	    REGION Part_MC_to_Robot
	        CASE #Dispatcher["_Part_MC_to_Robot"] OF
	            0: //nothing to do
	                ;
	            10: //prepare mission data
	                IF "SqlCommands".sqlCommands[0] = '' THEN
	                    IF #Gripper_ID[1] = 0 AND #Gripper_ID[2] = 0 THEN
	                        //nessuna pinza a bordo: impossibile prelevare
	                        #Error := 16;
	                        #Dispatcher["_Part_MC_to_Robot"] := "_Part_MC_to_Robot" * 100 + 1;
	                    ELSIF #GripperOccuped[1] AND #GripperOccuped[2] THEN
	                        //nessun lato libero: impossibile prelevare
	                        #Error := 18;
	                        #Dispatcher["_Part_MC_to_Robot"] := "_Part_MC_to_Robot" * 100 + 1;
	                    ELSIF (#MCRequested = 1 AND "DB_MC1".io_in.viceOpened) THEN
	                        // MORSA APERTA = NESSUN PEZZO DA PRELEVARE (17/9).
	                        // La ganascia aperta non puo' trattenere niente: qualunque
	                        // cosa dicano i registri, in morsa non c'e' un pezzo. Il
	                        // contrario NON vale — chiusa non implica pieno, puo'
	                        // essersi chiusa a vuoto — quindi il segnale si usa solo
	                        // come VETO, mai come conferma.
	                        #Error := 894;
	                        #Dispatcher["_Part_MC_to_Robot"] := 894;
	                    ELSE
	                        // QUOTE DALLA VISTA COORDINATES_Z_MC (19/9): vedi nota al
	                        // 10 di Part_Robot_to_MC.
	                        // Z_PICK_MC = prelievo del FINITO, che puo' avere presa
	                        // diversa dal grezzo (15/9).
	                        #queryTemp := 'select P.X,P.Y,Z.Z_PICK_MC,P.X_ROT,P.Y_ROT,P.Z_ROT,P.APPROACH_TYPE,P.APPROACH_X,P.APPROACH_Y,P.APPROACH_Z from POSITION P,COORDINATES_Z_MC Z where P.PARENT=$'MC_1$' and ';
	                        IF #RemoteMode THEN
	                            IF #MCRequested = 1 AND "DB_MC1".order.ID > 0 THEN
	                                #queryTemp := CONCAT(IN1 := #queryTemp,
	                                                     IN2 := 'Z.ORDER_ID=',
	                                                     IN3 := "INT_TO_STRING_WITHOUT_SIGN"(DINT_TO_INT("DB_MC1".order.ID)));
	                            ELSE
	                                #Error := 936;
	                                #Dispatcher["_Part_MC_to_Robot"] := "_Part_MC_to_Robot" * 100 + 1;
	                            END_IF;
	                        ELSE
	                            // HMI (29): ordine attivo se presente, altrimenti il piu' recente
	                            IF "DB_MC1".order.ID > 0 THEN
	                                #queryTemp := CONCAT(IN1 := #queryTemp,
	                                                     IN2 := 'Z.ORDER_ID=',
	                                                     IN3 := "INT_TO_STRING_WITHOUT_SIGN"(DINT_TO_INT("DB_MC1".order.ID)));
	                            ELSE
	                                #queryTemp := CONCAT(IN1 := #queryTemp,
	                                                     IN2 := 'Z.MC=1 order by Z.ORDER_ID desc');
	                            END_IF;
	                        END_IF;

	                        IF #Error = 0 THEN
	                            #queryStartExecution := TRUE;
	                            #Dispatcher["_Part_MC_to_Robot"] := 20;
	                        END_IF;
	                    END_IF;
	                END_IF;

	            20:  //execute query
	                // PRESA IN CARICO VERIFICATA: SqlData e' un buffer unico condiviso,
	                // senza il confronto su sqlCommands[0] si legge la risposta di un
	                // altro richiedente — qui sarebbero le QUOTE DI PRELIEVO dalla morsa.
	                IF NOT "DB_executeQuery".readyForNextQuery
	                    AND "SqlCommands".sqlCommands[0] = #queryTemp THEN
	                    #Dispatcher["_Part_MC_to_Robot"] := 30;
	                END_IF;

	            30:  // wait for result DB -> prepare mission data
	                IF "DB_executeQuery".dataReady AND "DB_executeQuery".noData THEN
	                    // quote di prelievo non trovate: con FB6 corretto "zero righe"
	                    // non e' piu' dataError, va intercettato qui.
	                    "DB_executeQuery".readyForNextQuery := true;
	                    #Error := "_Part_MC_to_Robot" * 100 + 99;       //Error 899
	                    #Dispatcher["_Part_MC_to_Robot"] := "_Part_MC_to_Robot" * 100 + 99;
	                ELSIF "DB_executeQuery".dataReady AND NOT "DB_executeQuery".dataError THEN

	                    // X DI PRELIEVO + CORSA DELLA SPINTA: se il pezzo e' stato
	                    // spinto in battuta non sta piu' dove il deposito lo ha messo.
	                    // xPushOffsetMC vale zero quando la spinta non c'e' stata,
	                    // quindi il caso normale resta invariato.
	                    "DB_RobotMission"."X_Pick-Place" := ("SqlData".data.rows[0].col[0]) + #xPushOffsetMC;
	                    "DB_RobotMission"."Y_Pick-Place" := ("SqlData".data.rows[0].col[1]);
	                    "DB_RobotMission"."Z_Pick-Place" := ("SqlData".data.rows[0].col[2]);
	                    "DB_RobotMission"."XRot_Pick-Place" := ("SqlData".data.rows[0].col[3]);
	                    "DB_RobotMission"."YRot_Pick-Place" := ("SqlData".data.rows[0].col[4]);
	                    "DB_RobotMission"."ZRot_Pick-Place" := ("SqlData".data.rows[0].col[5]);
	                    "DB_RobotMission".X_approach := ("SqlData".data.rows[0].col[7]);
	                    "DB_RobotMission".Y_approach := ("SqlData".data.rows[0].col[8]);
	                    "DB_RobotMission".Z_approach := ("SqlData".data.rows[0].col[9]);
	                    "DB_RobotMission".XRot_approach := 0;
	                    "DB_RobotMission".YRot_approach := 0;
	                    "DB_RobotMission".ZRot_approach := 0;
	                    //"DB_RobotMission".ApproachType := DINT_TO_INT("SqlData".data.rows[0].col[6]);
	                    "DB_RobotMission".ApproachType := "FC_ExtractApproach"(approachVal := "SqlData".data.rows[0].col[6], pick := TRUE);
	                    "DB_RobotMission".Object_Type := "Part";
	                    "DB_RobotMission".Unit_code := #MCRequested + 10;
	                    "DB_RobotMission".Gripper_code := #GripperRequested;
	                    // LATO SEMPRE DECISO (5/10): mancava l'ELSE. Con la doppia e il lato 2
	                    // pieno, o con la singola piena, Gripper_Side restava quello della
	                    // missione precedente e il robot prelevava con un lato occupato. Il lato
	                    // 1 della doppia e' del grezzo: il finito non ci va.
	                    "DB_executeQuery".readyForNextQuery := true;
	                    IF (#Gripper_ID[2] <> 0 AND NOT #GripperOccuped[2]) THEN
	                        "DB_RobotMission".Gripper_Side := 2;
	                        #Dispatcher["_Part_MC_to_Robot"] := 37;
	                    ELSIF (#Gripper_ID[2] = 0 AND #Gripper_ID[1] <> 0 AND NOT #GripperOccuped[1]) THEN
	                        "DB_RobotMission".Gripper_Side := 1;
	                        #Dispatcher["_Part_MC_to_Robot"] := 37;
	                    ELSE
	                        #Error := 18;   // nessun lato libero adatto al finito
	                        #Dispatcher["_Part_MC_to_Robot"] := "_Part_MC_to_Robot" * 100 + 1;
	                    END_IF;
	                    //"DB_RobotMission".Option
	                ELSIF "DB_executeQuery".dataError THEN
	                    "DB_executeQuery".readyForNextQuery := true;

	                    //Errore
	                    #Error := "_Part_MC_to_Robot" * 100 + 99;       //Error 899
	                    #Dispatcher["_Part_MC_to_Robot"] := "_Part_MC_to_Robot" * 100 + 99;
	                END_IF;

	            37:  // SOFFIAGGIO: vedi nota estesa al 37 di Part_Robot_to_MC.
	                // NB: qui X_Pick-Place e' la quota di PRELIEVO, che include
	                // xPushOffsetMC se il pezzo e' stato spinto. L'appoggio va
	                // calcolato sulla quota di DEPOSITO, quindi si sottrae l'offset
	                // per tornare alla nominale.
	                IF "SqlCommands".sqlCommands[0] = '' THEN
	                    IF "DB_MC1".order.ID > 0 THEN
	                        #queryTemp := CONCAT(IN1 := 'select CLAW_LENGTH,PART_WIDTH,STOP_BEYOND_CLAW from COORDINATES_BLOW_MC where ORDER_ID=',
	                                             IN2 := "INT_TO_STRING_WITHOUT_SIGN"(DINT_TO_INT("DB_MC1".order.ID)));
	                        #queryStartExecution := TRUE;
	                        #Dispatcher["_Part_MC_to_Robot"] := 38;
	                    ELSE
	                        #Dispatcher["_Part_MC_to_Robot"] := 40;
	                    END_IF;
	                END_IF;

	            38:  // presa in carico VERIFICATA
	                IF NOT "DB_executeQuery".readyForNextQuery
	                    AND "SqlCommands".sqlCommands[0] = #queryTemp THEN
	                    #Dispatcher["_Part_MC_to_Robot"] := 39;
	                END_IF;

	            39:  // esito: scrive le tre variabili PROFINET.
	                // APPOGGIO COME MISURA, NON COME QUOTA (19/9): il robotista non
	                // vuole piu' la posizione X del pezzo, che calcola per conto suo —
	                // gli serve solo di quanto il pezzo appoggia, cioe' meta' ganascia
	                // piu' il tratto oltre la ganascia dichiarato a pannello.
	                // Niente X_Pick-Place e niente xPushOffsetMC: l'offset serviva a
	                // riportare la quota di prelievo a quella di deposito, e senza la
	                // quota non ha piu' nulla da correggere. Sottraendolo dopo la
	                // divisione, per giunta, si toglievano MICRON da un numero in
	                // MILLIMETRI: col push attivo dava -49650.
	                IF "DB_executeQuery".dataReady THEN
	                    IF NOT "DB_executeQuery".noData AND NOT "DB_executeQuery".dataError THEN
	                        "Vice_ClawLength_mm" := DINT_TO_INT("SqlData".data.rows[0].col[0] / 1000);
	                        "Part_Width_mm" := DINT_TO_INT("SqlData".data.rows[0].col[1] / 1000);
	                        "X_Support_mm" := DINT_TO_INT(("SqlData".data.rows[0].col[0] / 2
	                                                                                    + "SqlData".data.rows[0].col[2]) / 1000);
	                    END_IF;
	                    "DB_executeQuery".readyForNextQuery := TRUE;
	                    #queryTemp := '';
	                    #queryStartExecution := FALSE;
	                    #Dispatcher["_Part_MC_to_Robot"] := 40;
	                END_IF;

	            40:
	                "DB_RobotMission".Command := "CMD_RobotPickObject";
	                IF "DB_RobotMissionStatus".StatusCode = "cmd_acquired" OR
	                    "DB_RobotMissionStatus".StatusCode = "cmd_executing" THEN
	                    #Dispatcher["_Part_MC_to_Robot"] := 50;
	                END_IF;
	            50:
	                IF "DB_RobotMissionStatus".StatusCode = "cmd_executed" THEN
	                    // lati dedicati: marca il lato realmente scelto (Gripper_Side: 1=grezzo, 2=finito)
	                    IF "DB_RobotMission".Gripper_Side = 2 THEN
	                        #GripperOccuped[2] := TRUE;
	                        #Dispatcher["updatePartOnRobot"] := 20 + DINT_TO_INT("FINISHED");
	                    ELSE
	                        #GripperOccuped[1] := TRUE;
	                        #Dispatcher["updatePartOnRobot"] := 10 + DINT_TO_INT("FINISHED");
	                    END_IF;
	                    "DB_RobotMission".Command := 0; ///\\\

	                    // Il pezzo spinto e' USCITO dalla macchina: la corsa memorizzata
	                    // non descrive piu' niente. Senza questo azzeramento resta
	                    // latchata e si somma al prelievo del pezzo SUCCESSIVO, che
	                    // magari non e' mai stato spinto.
	                    #xPushOffsetMC := 0;

	                    #Dispatcher["_Part_MC_to_Robot"] := 60;
	                END_IF;
	            60:
	                IF #Dispatcher["updatePartOnRobot"] = 0 THEN
	                    #Dispatcher["updatePartOnMC"] := 10 + DINT_TO_INT("EMPTY");
	                    IF #MCRequested = 1 THEN
	                        "DB_MC1".piecepresent[1] := 0;
	                    ELSIF #MCRequested = 2 THEN
	                        "DB_MC2".piecepresent[1] := 0;
	                    END_IF;

	                    #Dispatcher["_Part_MC_to_Robot"] := 70;
	                END_IF;
	            70:
	                IF #Dispatcher["updatePartOnMC"] = 0 THEN

	                    #Dispatcher["_Part_MC_to_Robot"] := 0;
	                END_IF;

	            894:
	                ; // morsa aperta: nessun pezzo da prelevare

	        END_CASE;
	    END_REGION

	END_REGION


	REGION TRAY_MANAGER
	    REGION TRAY_extact
	        CASE #Dispatcher["Extract_TRAY"] OF
	            0: //nothing to do
	                ;

	            10:
	                // GUARDIA PORTA OPERATORE (19/9): i cassetti non si muovono a
	                // porta aperta. Era l'unica catena del magazzino senza questo
	                // controllo — il comando estraeva il cassetto e il 949 arrivava
	                // dopo, a cassetto gia' fuori.
	                // Si legge l'ingresso direttamente: DB_BOX_1.Robot_enabled_to_work
	                // adesso dice solo "magazzino senza errori" e vale per pezzi e
	                // pinze, che a porta aperta possono proseguire.
	                IF NOT "Door_OP_locked" THEN
	                    #Error := 949;
	                    #Dispatcher["Extract_TRAY"] := 0;
	                ELSIF "DB_BOX_1".ExtractedTray = 0 THEN
	                    IF #Tray_ID > 0 AND #Tray_ID <= 12 THEN
	                        IF #Gripper_ID[1] = 0 AND #Gripper_ID[2] = 0 THEN
	                            #Error := 22;
	                            #Dispatcher["Extract_TRAY"] := 0;
	                        END_IF;
	                    ELSE
	                        #Error := 19001;
	                        // la catena chiude anche in errore (5/10): il parcheggio a 19001/19002
	                        // teneva il 750 fermo e MissionCode a 202 fino al reset
	                        #Dispatcher["Extract_TRAY"] := 0;
	                    END_IF;
	                ELSE
	                    IF "DB_BOX_1".ExtractedTray <> #Tray_ID THEN
	                        #Error := 19002;
	                        #Dispatcher["Extract_TRAY"] := 0;   // vedi nota al 19001
	                    END_IF;
	                END_IF;
	                IF #Dispatcher["Extract_TRAY"] = 10 THEN
	                    #Dispatcher["Extract_TRAY"] := 12;   // gancio già a bordo: nessun cambio-TCP
	                END_IF;

	            11: //wait for change TCP data
	                IF #Dispatcher["get_TCP_Data"] = 0 THEN
	                    #Dispatcher["Extract_TRAY"] := 12;
	                END_IF;

	            12:
	                IF "SqlCommands".sqlCommands[0] = '' AND "DB_executeQuery".readyForNextQuery THEN
	                    IF #Tray_ID > 0 AND #Tray_ID <> "DB_BOX_1".ExtractedTray THEN
	                        #queryTemp := CONCAT(IN1 := 'SELECT TRAY,X,Y,Z,X_ROT,Y_ROT,Z_ROT,APPROACH_TYPE,APPROACH_X,APPROACH_Y,APPROACH_Z from COORDINATES_FOR_EXTRACT where tray=',
	                                             IN2 := "INT_TO_STRING_WITHOUT_SIGN"(#Tray_ID));
	                        #queryStartExecution := TRUE;
	                        #Dispatcher["Extract_TRAY"] := 15;
	                    ELSIF #Tray_ID > 0 AND #Tray_ID = "DB_BOX_1".ExtractedTray THEN
	                        // IL CASSETTO CHIESTO E' GIA' FUORI (18/9): niente da fare,
	                        // la missione e' conclusa. Senza questo ramo la condizione
	                        // sopra e' falsa, il 12 non compone nessuna query e non
	                        // avanza: la catena resta appesa qui per sempre, il 750
	                        // aspetta Extract_TRAY=0 che non arriva mai e MissionCode
	                        // resta a 202 — con FB204 fermo al 58 in attesa di una
	                        // missione che nessuno chiudera'. Visto in campo.
	                        #Dispatcher["Extract_TRAY"] := 0;
	                    END_IF;
	                END_IF;

	            15:  // execute query — PRESA IN CARICO VERIFICATA
	                // SqlData e' un buffer unico condiviso: senza il confronto su
	                // sqlCommands[0] il 30 puo' leggere la risposta di un altro
	                // richiedente e mandare il robot a estrarre il cassetto con
	                // coordinate altrui.
	                IF NOT "DB_executeQuery".readyForNextQuery
	                    AND "SqlCommands".sqlCommands[0] = #queryTemp THEN
	                    #queryStartExecution := false;
	                    #Dispatcher["Extract_TRAY"] := 20;
	                END_IF;

	            20:  // wait result
	                // ZERO RIGHE = CASSETTO SENZA QUOTE (5/10). Con FB6 corretto "zero
	                // righe" non e' dataError: il 30 leggeva rows[0] rimasto dalla query
	                // PRECEDENTE e il robot andava a estrarre con quote altrui. Dopo le
	                // cancellazioni del 29/9 e' un caso reale.
	                IF "DB_executeQuery".dataReady AND NOT "DB_executeQuery".dataError
	                    AND NOT "DB_executeQuery".noData THEN
	                    #Dispatcher["Extract_TRAY"] := 30;
	                ELSIF "DB_executeQuery".dataReady AND NOT "DB_executeQuery".dataError THEN
	                    #Error := 19004;   // nessuna riga in COORDINATES_FOR_EXTRACT per il cassetto
	                    "DB_executeQuery".readyForNextQuery := TRUE;
	                    #queryTemp := '';
	                    #Dispatcher["Extract_TRAY"] := 0;
	                ELSIF "DB_executeQuery".dataReady AND "DB_executeQuery".dataError THEN
	                    #Error := 99; //DB ERROR
	                    "DB_executeQuery".readyForNextQuery := TRUE;
	                    #Dispatcher["Extract_TRAY"] := 0;
	                END_IF;

	            30: // prepare mission data for robot
	                IF NOT #GripperOccuped[1] AND NOT #GripperOccuped[2] THEN
	                    "DB_RobotMission"."X_Pick-Place" := "SqlData".data.rows[0].col[1];
	                    "DB_RobotMission"."Y_Pick-Place" := "SqlData".data.rows[0].col[2];
	                    "DB_RobotMission"."Z_Pick-Place" := "SqlData".data.rows[0].col[3];
	                    "DB_RobotMission"."XRot_Pick-Place" := "SqlData".data.rows[0].col[4];
	                    "DB_RobotMission"."YRot_Pick-Place" := "SqlData".data.rows[0].col[5];
	                    "DB_RobotMission"."ZRot_Pick-Place" := "SqlData".data.rows[0].col[6];
	                    "DB_RobotMission".X_approach := "SqlData".data.rows[0].col[8];
	                    "DB_RobotMission".Y_approach := "SqlData".data.rows[0].col[9];
	                    "DB_RobotMission".Z_approach := "SqlData".data.rows[0].col[10];
	                    "DB_RobotMission".XRot_approach := 0;
	                    "DB_RobotMission".YRot_approach := 0;
	                    "DB_RobotMission".ZRot_approach := 0;
	                    //"DB_RobotMission".ApproachType := DINT_TO_INT("SqlData".data.rows[0].col[7]);
	                    "DB_RobotMission".ApproachType := "FC_ExtractApproach"(approachVal := "SqlData".data.rows[0].col[7], pick := TRUE);
	                    "DB_RobotMission".Gripper_Side := 1;        //ALWAYS =1
	                    "DB_RobotMission".Object_Type := "TRAY";
	                    "DB_RobotMission".Unit_code := "Warehouse1";
	                    "DB_RobotMission".Gripper_code := #Gripper_ID[1];   // la pinza a bordo, non GripperRequested
	                    //"DB_RobotMission".Option

	                    "DB_executeQuery".readyForNextQuery := TRUE;
	                    #Dispatcher["Extract_TRAY"] := 40;
	                ELSE
	                    //gripper occupata
	                    #Error := 21;
	                    "DB_executeQuery".readyForNextQuery := TRUE;
	                    #Dispatcher["Extract_TRAY"] := 0;
	                END_IF;
	            40: //start mission robot
	                "DB_RobotMission".Command := "CMD_RobotExtractTray";
	                IF "DB_RobotMissionStatus".StatusCode = "cmd_acquired" OR
	                    "DB_RobotMissionStatus".StatusCode = "cmd_executing" THEN
	                    "DB_executeQuery".readyForNextQuery := TRUE;
	                    #queryTemp := '';
	                    #Dispatcher["Extract_TRAY"] := 100;
	                END_IF;

	            100: // Update DB — LATCH A DOPPIA CONFERMA
	                // Non basta cmd_executed del robot: senza il riscontro del sensore
	                // il registro dice "estratto" con il cassetto dentro, e la
	                // sincronizzazione di DB_BOX_1 tenta la richiusura (RequestedTray:=0)
	                // generando errore 9 e 949 a catena.
	                IF "DB_RobotMissionStatus".StatusCode = "cmd_executed"
	                    AND "px_tray_in_position"
	                THEN
	                    "FC_MQTT"(insert := true,
	                              send := false,
	                              topic := 'FROM_PLANT/TRAY/BOX/EXTRACT',
	                              payload := STRING_TO_WSTRING("INT_TO_STRING_WITHOUT_SIGN"(#Tray_ID)));

	                    "DB_RobotMission".Command := 0;  ///\\\

	                    "DB_BOX_1".ExtractedTray := #Tray_ID;
	                    #Dispatcher["Reset_or_log_MissionData"] := 10;
	                    #Dispatcher["Extract_TRAY"] := 130;
	                END_IF;
	            130:
	                IF #Dispatcher["Reset_or_log_MissionData"] = 0 AND "DB_RobotMissionStatus".StatusCode = "cmd_waitingNewCmd" THEN
	                    "DB_RobotMission".Gripper_code := #Gripper_ID[1];   // re-assert dopo il reset (come swap 985)
	                    #Dispatcher["Extract_TRAY"] := 0;
	                END_IF;

	        END_CASE;
	    END_REGION

	    REGION TRAY_release
	        CASE #Dispatcher["Release_TRAY"] OF
	            0: //nothing to do
	                ;
	            10:
	                // GUARDIA PORTA OPERATORE (19/9): vedi nota al 10 di Extract_TRAY.
	                IF NOT "Door_OP_locked" THEN
	                    #Error := 949;
	                    #Dispatcher["Release_TRAY"] := 0;
	                ELSIF "DB_BOX_1".ExtractedTray > 0 THEN
	                    IF #Gripper_ID[1] = 0 AND #Gripper_ID[2] = 0 THEN
	                        #Error := 2022;                     // pinza assente
	                        #Dispatcher["Release_TRAY"] := 0;
	                    ELSE
	                        #Dispatcher["Release_TRAY"] := 12;  // gancio a bordo: nessun cambio-TCP -> query
	                    END_IF;
	                ELSE
	                    #Error := 20001;                        // nessun cassetto da rilasciare
	                    #Dispatcher["Release_TRAY"] := 0;
	                END_IF;

	            11: //wait for change TCP data
	                IF #Dispatcher["get_TCP_Data"] = 0 THEN
	                    #Dispatcher["Release_TRAY"] := 12;
	                END_IF;

	            12:
	                IF "SqlCommands".sqlCommands[0] = '' THEN
	                    #queryTemp := CONCAT(IN1 := 'SELECT X,Y,Z,X_ROT,Y_ROT,Z_ROT,APPROACH_TYPE,APPROACH_X,APPROACH_Y,APPROACH_Z from COORDINATES_FOR_EXTRACT where tray=',
	                                         IN2 := "INT_TO_STRING_WITHOUT_SIGN"("DB_BOX_1".ExtractedTray));
	                    IF #MCRequested = 1 THEN
	                        #paramsTemp[0] := DINT_TO_INT("DB_MC1".order.GRIPPER);
	                        #paramsTemp[1] := DINT_TO_INT(IN := "RAW");
	                        IF ("DB_MC1".Status = "FINISHED") THEN
	                            #paramsTemp[1] := DINT_TO_INT(IN := "FINISHED");
	                        END_IF;
	                    ELSIF #MCRequested = 2 THEN
	                        #paramsTemp[0] := DINT_TO_INT("DB_MC2".order.GRIPPER);
	                        #paramsTemp[1] := DINT_TO_INT(IN := "RAW");
	                        IF ("DB_MC2".Status = "FINISHED") THEN
	                            #paramsTemp[1] := DINT_TO_INT(IN := "FINISHED");
	                        END_IF;
	                    END_IF;
	                    #queryStartExecution := TRUE;
	                    #Dispatcher["Release_TRAY"] := 15;
	                END_IF;

	            15: // execute query — PRESA IN CARICO VERIFICATA
	                // SqlData e' un buffer unico condiviso: senza il confronto su
	                // sqlCommands[0] il 30 puo' leggere la risposta di un altro
	                // richiedente e mandare il robot a rimettere dentro il cassetto
	                // con coordinate altrui.
	                IF NOT "DB_executeQuery".readyForNextQuery
	                    AND "SqlCommands".sqlCommands[0] = #queryTemp THEN
	                    #Dispatcher["Release_TRAY"] := 20;
	                END_IF;

	            20: // wait result
	                // ZERO RIGHE (5/10): vedi nota al 20 di Extract_TRAY. Qui il cassetto
	                // rientrerebbe con le quote di un altro.
	                // L'errore DB adesso chiude la catena (era parcheggiata a 99): l'810
	                // aspetta Release_TRAY = 0 e senza chiusura MissionCode restava a 203.
	                IF "DB_executeQuery".dataReady AND NOT "DB_executeQuery".dataError
	                    AND NOT "DB_executeQuery".noData THEN
	                    #Dispatcher["Release_TRAY"] := 30;
	                ELSIF "DB_executeQuery".dataReady AND NOT "DB_executeQuery".dataError THEN
	                    #Error := 20009;   // nessuna riga in COORDINATES_FOR_EXTRACT per il cassetto estratto
	                    "DB_executeQuery".readyForNextQuery := TRUE;
	                    #queryTemp := '';
	                    #Dispatcher["Release_TRAY"] := 0;
	                ELSIF "DB_executeQuery".dataError THEN
	                    #Error := 99;
	                    "DB_executeQuery".readyForNextQuery := TRUE;
	                    #Dispatcher["Release_TRAY"] := 0;
	                END_IF;

	            30:  // prepare mission data
	                IF NOT #GripperOccuped[1] AND NOT #GripperOccuped[2] THEN
	                    "DB_RobotMission"."X_Pick-Place" := "SqlData".data.rows[0].col[0];
	                    "DB_RobotMission"."Y_Pick-Place" := "SqlData".data.rows[0].col[1];
	                    "DB_RobotMission"."Z_Pick-Place" := "SqlData".data.rows[0].col[2];
	                    "DB_RobotMission"."XRot_Pick-Place" := "SqlData".data.rows[0].col[3];
	                    "DB_RobotMission"."YRot_Pick-Place" := "SqlData".data.rows[0].col[4];
	                    "DB_RobotMission"."ZRot_Pick-Place" := "SqlData".data.rows[0].col[5];
	                    "DB_RobotMission".X_approach := "SqlData".data.rows[0].col[7];
	                    "DB_RobotMission".Y_approach := "SqlData".data.rows[0].col[8];
	                    "DB_RobotMission".Z_approach := "SqlData".data.rows[0].col[9];
	                    "DB_RobotMission".XRot_approach := 0;
	                    "DB_RobotMission".YRot_approach := 0;
	                    "DB_RobotMission".ZRot_approach := 0;
	                    //"DB_RobotMission".ApproachType := DINT_TO_INT("SqlData".data.rows[0].col[6]);
	                    "DB_RobotMission".ApproachType := "FC_ExtractApproach"(approachVal := "SqlData".data.rows[0].col[6], pick := TRUE);
	                    "DB_RobotMission".Object_Type := "TRAY";
	                    "DB_RobotMission".Gripper_Side := 1; //ALWAYS 1
	                    "DB_RobotMission".Unit_code := "Warehouse1";
	                    "DB_RobotMission".Gripper_code := #Gripper_ID[1];   // la pinza a bordo, non GripperRequested
	                    //"DB_RobotMission".Option

	                    "DB_executeQuery".readyForNextQuery := TRUE;
	                    #Dispatcher["Release_TRAY"] := 40;
	                ELSE
	                    //gripper occupata
	                    #Error := 21;
	                    "DB_executeQuery".readyForNextQuery := TRUE;
	                    #Dispatcher["Release_TRAY"] := 0;
	                END_IF;
	            40:
	                "DB_RobotMission".Command := "CMD_RobotReleaseTray";
	                IF "DB_RobotMissionStatus".StatusCode = "cmd_acquired" OR
	                    "DB_RobotMissionStatus".StatusCode = "cmd_executing" THEN
	                    "DB_executeQuery".readyForNextQuery := TRUE;
	                    #queryTemp := '';
	                    #Dispatcher["Release_TRAY"] := 100;
	                END_IF;

	            100: // Update DB -----------------------------------------
	                IF "DB_RobotMissionStatus".StatusCode = "cmd_executed" THEN
	                    "FC_MQTT"(insert := true,
	                              send := false,
	                              topic := 'FROM_PLANT/TRAY/BOX/RELEASE',
	                              payload := STRING_TO_WSTRING("INT_TO_STRING_WITHOUT_SIGN"("DB_BOX_1".ExtractedTray)));
	                    "DB_RobotMission".Command := 0;  ///\\\
	                    "DB_BOX_1".ExtractedTray := 0;
	                    #Dispatcher["Reset_or_log_MissionData"] := 10;
	                    #Dispatcher["Release_TRAY"] := 130;
	                END_IF;
	                (*
	                   IF "DB_RobotMissionStatus".StatusCode = "cmd_executed" THEN#paramsTemp[0] := 0;
	                    #paramsTemp[1] := "DB_BOX_1".ExtractedTray;

	                    #Dispatcher["Release_TRAY"] := 105;
	                END_IF;
	            105: //wait for DB ready
	                IF "DB_executeQuery".readyForNextQuery THEN
	                    #Dispatcher["Release_TRAY"] := 110;
	                END_IF;
	            110:  // execute query
	                IF NOT "DB_executeQuery".readyForNextQuery THEN
	                    #Dispatcher["Release_TRAY"] := 120;
	                END_IF;

	            120:  // wait result
	                IF "DB_executeQuery".dataReady  THEN //AND NOT "DB_executeQuery".dataError
	                    "DB_BOX_1".ExtractedTray := 0;
	                    "DB_executeQuery".readyForNextQuery := TRUE;

	                    #Dispatcher["Reset_or_log_MissionData"] := 10;

	                    #Dispatcher["Release_TRAY"] := 130;
	                END_IF;
	            *)
	            130:
	                IF #Dispatcher["Reset_or_log_MissionData"] = 0 AND "DB_RobotMissionStatus".StatusCode = "cmd_waitingNewCmd" THEN
	                    "DB_RobotMission".Gripper_code := #Gripper_ID[1];
	                    #Dispatcher["Release_TRAY"] := 0;
	                END_IF;
	        END_CASE;
	    END_REGION
	END_REGION

	REGION MICROMISSIONS_AND_UPDATE_DB
	    REGION get_TCP_Data
	        CASE #Dispatcher["get_TCP_Data"] OF
	            0: //nothing to do
	                ;
	            10: //prepare mission data ***START HERE FOR GRIPPER***
	                IF "SqlCommands".sqlCommands[0] = '' THEN
	                    IF #Gripper_ID[1] = 0 AND #Gripper_ID[2] = 0 THEN
	                        //gripper absent
	                        #Error := "get_TCP_Data" * 100 + 22;        //error 2222
	                        #Dispatcher["get_TCP_Data"] := 0;
	                    ELSE
	                        #queryTemp := 'tcpData';
	                        #queryStartExecution := TRUE;

	                        #Dispatcher["get_TCP_Data"] := 15;
	                    END_IF;
	                END_IF;
	            12: //prepare mission data ***START HERE FOR HOOK***
	                IF "SqlCommands".sqlCommands[0] = '' THEN
	                    IF #Gripper_ID[1] = 0 AND #Gripper_ID[2] = 0 THEN
	                        //gripper absent
	                        #Error := 22;
	                        #Dispatcher["get_TCP_Data"] := 0;
	                    ELSE
	                        #queryTemp := 'select X,Y,Z,0,X_ROT,Y_ROT,Z_ROT from GRIPPER_HOOK';  //la colonna 4 (0) serve solo per tenere il posto vuoto della valvola ottenuta con l'altra query
	                        #queryStartExecution := TRUE;

	                        #Dispatcher["get_TCP_Data"] := 15;
	                    END_IF;
	                END_IF;

	            15: //wait DB ready — PRESA IN CARICO VERIFICATA
	                // SqlData e' un buffer unico condiviso: senza verifica il 30 puo'
	                // leggere la risposta di un altro richiedente e mandare al robot
	                // dimensioni TCP sbagliate.
	                // 'tcpData' e' una query SPECIALE che FB6 espande: sqlCommands[0] non
	                // coincide mai con #queryTemp, quindi la presa in carico si riconosce
	                // dall'inizio della query espansa. Sul ramo del gancio (stato 12) la
	                // query e' letterale e il confronto diretto vale.
	                // 5/10: a presa in carico avvenuta il flag si abbassa QUI, perche' per
	                // 'tcpData' OB1 rete 7 non lo abbassa mai: col ponte condiviso il
	                // robot terrebbe la precedenza per sempre e FB204 non potrebbe piu'
	                // interrogare il DB.
	                IF NOT "DB_executeQuery".readyForNextQuery THEN
	                    IF (#queryTemp = 'tcpData'
	                        AND LEFT(IN := "SqlCommands".sqlCommands[0], L := 20) = 'select X_BODY+X_CLAW')
	                        OR (#queryTemp <> 'tcpData'
	                        AND "SqlCommands".sqlCommands[0] = #queryTemp)
	                    THEN
	                        #queryStartExecution := FALSE;
	                        #Dispatcher["get_TCP_Data"] := 20;
	                    END_IF;
	                END_IF;

	            20: //wait answer
	                // ZERO RIGHE PRIMA DEL SUCCESSO (5/10). Il ramo noData stava dopo quello
	                // di successo, che e' vero anche con zero righe: era irraggiungibile, e
	                // il 30 mandava al robot le dimensioni TCP della query precedente.
	                // La ricerca gancio (22-26, TODO mai finito) non parte piu' da qui:
	                // pinza a bordo assente dal database = errore dichiarato.
	                IF "DB_executeQuery".dataReady AND NOT "DB_executeQuery".dataError
	                    AND "DB_executeQuery".noData THEN
	                    "DB_executeQuery".readyForNextQuery := TRUE;
	                    #queryTemp := '';
	                    #queryStartExecution := FALSE;
	                    #Error := 2205;   // pinza a bordo assente da GRIPPERS / GRIPPER_HOOK
	                    #Dispatcher["get_TCP_Data"] := 0;
	                ELSIF "DB_executeQuery".dataReady AND NOT "DB_executeQuery".dataError THEN
	                    #Dispatcher["get_TCP_Data"] := 30;
	                ELSIF "DB_executeQuery".dataError THEN
	                    // chiusura anche in errore DB (5/10): il parcheggio a 99 lasciava
	                    // appesi i chiamanti (120, 960, 980, Declare 50) fino al reset
	                    "DB_executeQuery".readyForNextQuery := true; //****
	                    #Error := 99;
	                    #Dispatcher["get_TCP_Data"] := 0;
	                END_IF;

	            22:
	                IF #Dispatcher["_Gripper_Hook_Search"] = 0 THEN
	                    #Dispatcher["_Gripper_Robot_to_TRAY"] := 10;
	                    #Dispatcher["get_TCP_Data"] := 24;
	                END_IF;
	            24:
	                IF #Dispatcher["_Gripper_Robot_to_TRAY"] = 0 THEN
	                    #MCRequested := 0;
	                    #Dispatcher["_Gripper_TRAY_to_Robot"] := 10;
	                    #Dispatcher["get_TCP_Data"] := 26;
	                END_IF;
	            26:
	                IF #Dispatcher["_Gripper_TRAY_to_Robot"] = 0 THEN
	                    #GripperRequested := 0;
	                    #Dispatcher["get_TCP_Data"] := 12;
	                END_IF;


	            30:  // wait for result DB -> prepare mission data
	                "DB_RobotMission".Gripper1_XDim := "SqlData".data.rows[0].col[0];
	                "DB_RobotMission".Gripper1_YDim := "SqlData".data.rows[0].col[1];
	                "DB_RobotMission".Gripper1_ZDim := "SqlData".data.rows[0].col[2];
	                "DB_RobotMission".Gripper1_XRotDim := "SqlData".data.rows[0].col[4];
	                "DB_RobotMission".Gripper1_YRotDim := "SqlData".data.rows[0].col[5];
	                "DB_RobotMission".Gripper1_ZRotDim := "SqlData".data.rows[0].col[6];
	                "DB_RobotMission".Gripper_code := #Gripper_ID[1]; //???

	                IF "SqlData".data.rowCount > 1 THEN
	                    // lato 2: dimensioni dalla riga gemella.
	                    // Le ROTAZIONI del lato 2 le gestisce il robot con il proprio TCP:
	                    // il PLC non le manda e le tiene a zero per non lasciare valori
	                    // stantii (il calcolo +180 del 2/9 produceva 270000 e falsava tutto).
	                    "DB_RobotMission".Gripper2_XDim := "SqlData".data.rows[1].col[0];
	                    "DB_RobotMission".Gripper2_YDim := "SqlData".data.rows[1].col[1];
	                    "DB_RobotMission".Gripper2_ZDim := "SqlData".data.rows[1].col[2];
	                    "DB_RobotMission".Gripper2_XRotDim := 0;
	                    "DB_RobotMission".Gripper2_YRotDim := 0;
	                    "DB_RobotMission".Gripper2_ZRotDim := 0;
	                    "DB_RobotMission".Gripper_code := #Gripper_ID[2]; //???
	                END_IF;

	                #i := DINT_TO_INT("SqlData".data.rows[0].col[3]);
	                IF #i > 10 THEN
	                    "DB_RobotMission".Gripper1_Valve := #i - DINT_TO_INT(TRUNC(#i / 10) * 10);
	                    "DB_RobotMission".Gripper2_Valve := TRUNC(#i / 10);
	                ELSE
	                    "DB_RobotMission".Gripper1_Valve := #i;
	                    "DB_RobotMission".Gripper2_Valve := 0;
	                END_IF;

	                "DB_executeQuery".readyForNextQuery := true;
	                #Dispatcher["get_TCP_Data"] := 40;

	            40: //sync with robot
	                IF "DB_RobotMissionStatus".StatusCode = "cmd_waitingNewCmd" THEN  ////\\\\
	                    #Dispatcher["get_TCP_Data"] := 45;
	                END_IF;
	            45: // Robot execute mission
	                "DB_RobotMission".Command := "CMD_RobotChangeDataForGripper";
	                IF "DB_RobotMissionStatus".StatusCode = "cmd_acquired" OR
	                    "DB_RobotMissionStatus".StatusCode = "cmd_executing" THEN
	                    #Dispatcher["get_TCP_Data"] := 50;
	                END_IF;

	            50:  // robot end mission
	                IF "DB_RobotMissionStatus".StatusCode = "cmd_executed" THEN
	                    "DB_RobotMission".Command := 0;  ///\\\
	                    "DB_executeQuery".readyForNextQuery := true;

	                    #Dispatcher["get_TCP_Data"] := 55;
	                END_IF;
	            55:
	                #Dispatcher["updateGripperOnRobot"] := 10; //serve fare questo?? TODO

	                #Dispatcher["get_TCP_Data"] := 100;
	            100:
	                IF #Dispatcher["updateGripperOnRobot"] = 0 THEN
	                    //"DB_executeQuery".readyForNextQuery := true;  //paolo 18/8

	                    #Dispatcher["Reset_or_log_MissionData"] := 10;
	                    #Dispatcher["get_TCP_Data"] := 110;
	                END_IF;
	            110:
	                IF #Dispatcher["Reset_or_log_MissionData"] = 0 AND "DB_RobotMissionStatus".StatusCode = 0 THEN
	                    #Dispatcher["get_TCP_Data"] := 0;
	                END_IF;
	        END_CASE;
	    END_REGION

	    REGION updateGripperOnRobot
	        CASE #Dispatcher["updateGripperOnRobot"] OF
	            0:  // nothing to do
	                ;
	            10: // Update DB ***START HERE***
	                IF "SqlCommands".sqlCommands[0] = '' THEN
	                    IF #Gripper_ID[1] > 0 AND #Gripper_ID[2] > 0 THEN
	                        // pinza a doppia presa: entrambe le righe gemelle a bordo.
	                        // NB: niente IN(...) — il ponte SQL non lo digerisce e resta appeso.
	                        #queryTemp := CONCAT(IN1 := 'UPDATE GRIPPER SET POS_PLANT = 0 WHERE POS_plant = 1000; ',
	                                             IN2 := 'UPDATE Gripper SET POS_PLANT=1000 WHERE ID = ',
	                                             IN3 := "INT_TO_STRING_WITHOUT_SIGN"(#Gripper_ID[1]),
	                                             IN4 := '; UPDATE Gripper SET POS_PLANT=1000 WHERE ID = ',
	                                             IN5 := "INT_TO_STRING_WITHOUT_SIGN"(#Gripper_ID[2]));
	                    ELSIF #Gripper_ID[1] > 0 THEN
	                        #queryTemp := CONCAT(IN1 := 'UPDATE GRIPPER SET POS_PLANT = 0 WHERE POS_plant = 1000; ',
	                                             IN2 := 'UPDATE Gripper SET POS_PLANT=1000 WHERE ID = ',
	                                             IN3 := "INT_TO_STRING_WITHOUT_SIGN"(#Gripper_ID[1]));
	                    ELSE
	                        #queryTemp := 'UPDATE GRIPPER SET POS_PLANT=0 WHERE POS_PLANT=1000';
	                    END_IF;
	                    #queryStartExecution := TRUE;

	                    #Dispatcher["updateGripperOnRobot"] := 20;
	                END_IF;

	            20:  // execute query
	                IF NOT "DB_executeQuery".readyForNextQuery THEN
	                    #Dispatcher["updateGripperOnRobot"] := 30;
	                END_IF;

	            30:  // wait result
	                IF "DB_executeQuery".dataReady THEN

	                    "DB_executeQuery".readyForNextQuery := TRUE;
	                    #Dispatcher["updateGripperOnRobot"] := 0;

	                    "FC_MQTT"(insert := true,
	                              send := false,
	                              topic := 'FROM_PLANT/GRIPPER/ROBOT',
	                              payload := STRING_TO_WSTRING("INT_TO_STRING_WITHOUT_SIGN"(#Gripper_ID[1])));

	                ELSIF "DB_executeQuery".dataError THEN
	                    // Alarm
	                    #Error := 99;
	                    #Dispatcher["updateGripperOnRobot"] := 99;
	                END_IF;
	        END_CASE;
	    END_REGION

	    REGION updatePartOnRobot
	        CASE #Dispatcher["updatePartOnRobot"] OF
	            0:  // nothing to do
	                ;

	            10..15: // Update DB ------------ *** START HERE *** (change status Gripper 1)
	                IF "SqlCommands".sqlCommands[0] = '' THEN
	                    //la attivo con dispatcher=10+statoPezzo (RAW,FINISHED)
	                    (* Modificato il 16/09/2025
	                    IF #GripperOccuped[1] THEN
	                        #queryTemp := CONCAT(IN1 := 'UPDATE GRIPPER SET STATUS=',
	                                             IN2 := "INT_TO_STRING_WITHOUT_SIGN"(#Dispatcher["updatePartOnRobot"] - 10),
	                                             IN3 := ' WHERE ID=',
	                                             IN4 := "INT_TO_STRING_WITHOUT_SIGN"(#Gripper_ID[1]));
	                    ELSE
	                        #queryTemp := CONCAT(IN1 := 'UPDATE GRIPPER SET STATUS=2 WHERE ID=',    //EMPTY
	                                             IN2 := "INT_TO_STRING_WITHOUT_SIGN"(#Gripper_ID[1]));
	                    END_IF;
	                    *)
	                    #queryTemp := CONCAT(IN1 := 'UPDATE GRIPPER SET STATUS=',
	                                         IN2 := "INT_TO_STRING_WITHOUT_SIGN"(#Dispatcher["updatePartOnRobot"] - 10),
	                                         IN3 := ' WHERE ID=',
	                                         IN4 := "INT_TO_STRING_WITHOUT_SIGN"(#Gripper_ID["DB_RobotMission".Gripper_Side]));

	                    #queryStartExecution := true;
	                    #Dispatcher["updatePartOnRobot"] := 40;
	                END_IF;

	            20..25: // Update DB ------------ *** START HERE *** (change status gripper 2)
	                IF "SqlCommands".sqlCommands[0] = '' THEN
	                    //la attivo con dispatcher=20+statoPezzo (RAW,FINISHED)
	                    IF #GripperOccuped[2] THEN
	                        #queryTemp := CONCAT(IN1 := 'UPDATE GRIPPER SET STATUS=',
	                                             IN2 := "INT_TO_STRING_WITHOUT_SIGN"(#Dispatcher["updatePartOnRobot"] - 20),
	                                             IN3 := ' WHERE ID=',
	                                             IN4 := "INT_TO_STRING_WITHOUT_SIGN"(#Gripper_ID[2]));
	                    ELSE
	                        #queryTemp := CONCAT(IN1 := 'UPDATE GRIPPER SET STATUS=2 WHERE ID=',    //EMPTY
	                                             IN2 := "INT_TO_STRING_WITHOUT_SIGN"(#Gripper_ID[2]));
	                    END_IF;

	                    #queryStartExecution := true;
	                    #Dispatcher["updatePartOnRobot"] := 40;
	                END_IF;

	            40:  // execute query
	                IF NOT "DB_executeQuery".readyForNextQuery THEN
	                    #Dispatcher["updatePartOnRobot"] := 50;
	                END_IF;

	            50:  // wait result
	                IF "DB_executeQuery".dataReady THEN
	                    "DB_executeQuery".readyForNextQuery := TRUE;

	                    #Dispatcher["updatePartOnRobot"] := 55;
	                END_IF;

	            55:// wait for reset query
	                IF "DB_executeQuery".Dispatch["_master"] = 0 AND "SqlCommands".sqlCommands[0] = '' THEN
	                    "FC_MQTT"(insert := true,
	                              send := false,
	                              topic := 'FROM_PLANT/GRIPPER/ROBOT',
	                              payload := STRING_TO_WSTRING("INT_TO_STRING_WITHOUT_SIGN"(#Gripper_ID[1])));

	                    #Dispatcher["updatePartOnRobot"] := 0;
	                END_IF;

	        END_CASE;
	    END_REGION

	    REGION updatePalletOnTRAY
	        CASE #Dispatcher["updatePalletOnTRAY"] OF
	            0:  // nothing to do
	                ;

	            10..15: // *** START HERE *** (change status)
	                IF "SqlCommands".sqlCommands[0] = '' THEN
	                    //la attivo con dispatcher=10+statoPezzo (RAW,FINISHED)
	                    IF #GripperOccuped[1] THEN
	                        //robot finish a pick
	                        #queryTemp := CONCAT(IN1 := 'UPDATE [POSITION] SET STATUS=',
	                                             IN2 := "INT_TO_STRING_WITHOUT_SIGN"(#Dispatcher["updatePalletOnTRAY"] - 10));
	                        IF #MCRequested = 0 THEN  //HMI command
	                            #queryTemp := CONCAT(IN1 := #queryTemp,
	                                                 IN2 := ' WHERE parent like $'WPALLET%$' AND SUB_POS = ',
	                                                 IN3 := "INT_TO_STRING_WITHOUT_SIGN"(#PalletPosition),
	                                                 IN4 := '; UPDATE Pallet SET POS_PLANT=1000 WHERE mag_pos=',
	                                                 IN5 := "INT_TO_STRING_WITHOUT_SIGN"(#PalletPosition));
	                            #queryStartExecution := true;
	                            #Dispatcher["updatePalletOnTRAY"] := 20;

	                        ELSIF #MCRequested = 1 AND "DB_MC1".order.ID > 0 THEN
	                            #queryTemp := CONCAT(IN1 := #queryTemp,
	                                                 IN2 := ' WHERE parent like $'WPALLET%$' AND SUB_POS in(select top 1 pos from COORDINATES_FOR_PALLET_WAREHOUSE where status=4 AND PalletID =  ',  //raw
	                                                 IN3 := "INT_TO_STRING_WITHOUT_SIGN"(DINT_TO_INT("DB_MC1".order.PALLET)),  // .order.ID   Order_ID ....
	                                                 IN4 := ')',
	                                                 IN5 := '; UPDATE Pallet SET POS_PLANT=1000 WHERE id=',
	                                                 IN6 := "INT_TO_STRING_WITHOUT_SIGN"(DINT_TO_INT("DB_MC1".order.PALLET)));
	                            #queryStartExecution := true;
	                            #Dispatcher["updatePalletOnTRAY"] := 20;

	                        ELSIF #MCRequested = 2 AND "DB_MC2".order.ID > 0 THEN
	                            #queryTemp := CONCAT(IN1 := #queryTemp,
	                                                 IN2 := ' WHERE parent like $'WPALLET%$' AND SUB_POS in (select top 1 pos from COORDINATES_FOR_PALLET_WAREHOUSE where status=4 AND PalletID =  ',  //raw
	                                                 IN3 := "INT_TO_STRING_WITHOUT_SIGN"(DINT_TO_INT("DB_MC2".order.PALLET)),
	                                                 IN4 := ')',
	                                                 IN5 := '; UPDATE Pallet SET POS_PLANT=1000 WHERE id=',
	                                                 IN6 := "INT_TO_STRING_WITHOUT_SIGN"(DINT_TO_INT("DB_MC2".order.PALLET)));
	                            #queryStartExecution := true;
	                            #Dispatcher["updatePalletOnTRAY"] := 20;
	                        END_IF;

	                    ELSE
	                        //robot finish a release on warehouse
	                        #queryTemp := CONCAT(IN1 := 'UPDATE [POSITION] SET STATUS=',
	                                             IN2 := "INT_TO_STRING_WITHOUT_SIGN"(#Dispatcher["updatePalletOnTRAY"] - 10)); //empty
	                        IF #MCRequested = 0 THEN  //HMI command
	                            #queryTemp := CONCAT(IN1 := #queryTemp,
	                                                 IN2 := ' WHERE parent like $'WPALLET%$' AND SUB_POS = ',
	                                                 IN3 := "INT_TO_STRING_WITHOUT_SIGN"(#PalletPosition),
	                                                 IN4 := '; UPDATE Pallet SET POS_PLANT=0 WHERE mag_pos=',
	                                                 IN5 := "INT_TO_STRING_WITHOUT_SIGN"(#PalletPosition));
	                            #queryStartExecution := true;
	                            #Dispatcher["updatePalletOnTRAY"] := 20;

	                        ELSIF #MCRequested = 1 AND "DB_MC1".order.ID > 0 THEN
	                            #queryTemp := CONCAT(IN1 := #queryTemp,
	                                                 IN2 := ' WHERE id in(select top 1 id from COORDINATES_FOR_PALLET_WAREHOUSE where status=2 AND PalletID= ', //empty
	                                                 IN3 := "INT_TO_STRING_WITHOUT_SIGN"(DINT_TO_INT("DB_MC1".order.PALLET)),
	                                                 IN4 := ')',
	                                                 IN5 := '; UPDATE Pallet SET POS_PLANT=0 WHERE id=',
	                                                 IN6 := "INT_TO_STRING_WITHOUT_SIGN"(#PalletRequested));
	                            #queryStartExecution := true;
	                            #Dispatcher["updatePalletOnTRAY"] := 20;

	                        ELSIF #MCRequested = 2 AND "DB_MC2".order.ID > 0 THEN
	                            #queryTemp := CONCAT(IN1 := #queryTemp,
	                                                 IN2 := ' WHERE id in(select top 1 id from COORDINATES_FOR_PALLET_WAREHOUSE where status=2 AND PalletID= ', //empty
	                                                 IN3 := "INT_TO_STRING_WITHOUT_SIGN"(DINT_TO_INT("DB_MC2".order.PALLET)),
	                                                 IN4 := ')',
	                                                 IN5 := '; UPDATE Pallet SET POS_PLANT=0 WHERE id=',
	                                                 IN6 := "INT_TO_STRING_WITHOUT_SIGN"(#PalletRequested));
	                            #queryStartExecution := true;
	                            #Dispatcher["updatePalletOnTRAY"] := 20;
	                        END_IF;

	                    END_IF;

	                END_IF;

	            20:  // execute query
	                IF NOT "DB_executeQuery".readyForNextQuery THEN
	                    #Dispatcher["updatePalletOnTRAY"] := 30;
	                END_IF;

	            30:  // wait result
	                IF "DB_executeQuery".dataReady THEN
	                    "DB_executeQuery".readyForNextQuery := TRUE;

	                    #Dispatcher["updatePalletOnTRAY"] := 35;
	                END_IF;

	            35:// wait for reset query
	                IF "DB_executeQuery".Dispatch["_master"] = 0 AND "SqlCommands".sqlCommands[0] = '' THEN
	                    #Dispatcher["updatePalletOnTRAY"] := 0;
	                END_IF;

	        END_CASE;
	    END_REGION

	    REGION updatePartOnMC
	        //la attivo con dispatcher=10+statoPezzo (RAW,FINISHED)
	        CASE #Dispatcher["updatePartOnMC"] OF
	            0:  // nothing to do
	                ;

	            10..15: // Update DB -----------------------------------------
	                // NOT queryStartExecution (5/10): questa catena la lancia anche FB204
	                // (36, 37, 41, riconciliazione al 50), in modo asincrono. Se nello
	                // stesso scan un'altra catena di FB7 ha appena composto la sua query,
	                // il ponte e' ancora vuoto ma queryTemp e' occupato: non va sovrascritto.
	                IF "SqlCommands".sqlCommands[0] = '' AND NOT #queryStartExecution THEN
	                    #pieceReq := DINT_TO_INT("DB_MC1".order.PIECE);
	                    IF (#MCRequested = 2) THEN
	                        #pieceReq := DINT_TO_INT("DB_MC2".order.PIECE);
	                    END_IF;
	                    // MACCHINA DI DEFAULT MC1 (5/10): a riposo MCRequested vale 0 e la
	                    // UPDATE andava su PARENT 'MC_0%', nessuna riga: il DB non seguiva i
	                    // comandi 36, 37 e 41 del pannello. La cella ha una sola macchina.
	                    #temp := #MCRequested;
	                    IF #temp <= 0 THEN
	                        #temp := 1;
	                    END_IF;
	                    #queryTemp := CONCAT(IN1 := 'UPDATE POSITION SET STATUS=',
	                                         IN2 := "INT_TO_STRING_WITHOUT_SIGN"(#Dispatcher["updatePartOnMC"] - 10),
	                                         IN3 := ' WHERE PARENT like $'MC_',
	                                         IN4 := "INT_TO_STRING_WITHOUT_SIGN"(#temp),
	                                         IN5 := '%$' AND PARENT NOT LIKE $'%pallet%$' ');  //AND Part_Type='
	                    //IN6 := "INT_TO_STRING_WITHOUT_SIGN"(#pieceReq));
	                    #queryStartExecution := TRUE;

	                    // REGISTRO PEZZO IN MACCHINA (5/10). EMPTY vuol dire vuota: registro
	                    // a zero. Prima si scriveva order.PIECE anche per EMPTY, e dopo un
	                    // prelievo il 60 di Part_MC_to_Robot azzerava il registro e qui
	                    // tornava subito "pieno".
	                    // Per RAW e FINISHED l'ordine si scrive SOLO a registro vuoto: un
	                    // valore gia' presente l'ha messo chi sa cosa c'e' in morsa (FB204
	                    // prima del deposito, la dichiarazione 36 dal pannello) e l'ordine,
	                    // a riposo, puo' valere zero o essere un altro.
	                    IF #temp = 1 THEN
	                        IF #Dispatcher["updatePartOnMC"] - 10 = DINT_TO_INT("EMPTY") THEN
	                            "DB_MC1".piecepresent[1] := 0;
	                        ELSIF "DB_MC1".piecepresent[1] = 0 THEN
	                            "DB_MC1".piecepresent[1] := DINT_TO_INT("DB_MC1".order.PIECE);
	                        END_IF;
	                    ELSIF #temp = 2 THEN
	                        IF #Dispatcher["updatePartOnMC"] - 10 = DINT_TO_INT("EMPTY") THEN
	                            "DB_MC2".piecepresent[1] := 0;
	                        ELSIF "DB_MC2".piecepresent[1] = 0 THEN
	                            "DB_MC2".piecepresent[1] := DINT_TO_INT("DB_MC2".order.PIECE);
	                        END_IF;
	                    END_IF;

	                    #Dispatcher["updatePartOnMC"] := 20;
	                END_IF;
	            20:  // execute query
	                IF NOT "DB_executeQuery".readyForNextQuery THEN
	                    #Dispatcher["updatePartOnMC"] := 30;
	                END_IF;

	            21..25: // deposito PALLET in macchina -> POS_PLANT=100+MC
	                // STATO DI LAVORO FUORI RANGE (17/9): questo ramo deve uscire dal
	                // proprio range prima di attendere il ponte. Prima, se
	                // sqlCommands[0] era occupata dalla query di un'altra catena, la
	                // guardia era falsa, il registro restava a 2x e NESSUNO lo faceva
	                // avanzare: il ramo e' il suo stesso stato di attesa, quindi non
	                // veniva mai piu' rivalutato con esito utile. Visto in campo col
	                // pallet appena montato: registro fermo a 24, query gia' nel ponte,
	                // catena morta e ciclo bloccato prima dello start lavorazione.
	                // Con il salto al 26 la composizione avviene una volta sola, quando
	                // il ponte e' libero, e l'attesa ha uno stato suo.
	                IF "SqlCommands".sqlCommands[0] = '' THEN
	                    IF NOT #RemoteMode THEN
	                        #pieceReq := #PalletRequested;
	                    ELSE
	                        #pieceReq := DINT_TO_INT("DB_MC1".order.PALLET);
	                    END_IF;
	                    #queryTemp := CONCAT(IN1 := 'UPDATE POSITION SET STATUS=',
	                                         IN2 := "INT_TO_STRING_WITHOUT_SIGN"(#Dispatcher["updatePartOnMC"] - 20),
	                                         IN3 := ' WHERE PARENT like $'MC_',
	                                         IN4 := "INT_TO_STRING_WITHOUT_SIGN"(#MCRequested),
	                                         IN5 := '%$' AND PARENT NOT LIKE $'%pallet%$'; UPDATE Pallet SET POS_PLANT=',
	                                         IN6 := "INT_TO_STRING_WITHOUT_SIGN"(100 + #MCRequested),
	                                         IN7 := ' WHERE ID=',
	                                         IN8 := "INT_TO_STRING_WITHOUT_SIGN"(#pieceReq));
	                    #queryStartExecution := TRUE;
	                    #Dispatcher["updatePartOnMC"] := 26;
	                END_IF;

	            26:  // attesa presa in carico della query pallet (stato fuori dai range)
	                IF NOT "DB_executeQuery".readyForNextQuery THEN
	                    #Dispatcher["updatePartOnMC"] := 30;
	                END_IF;

	            30:  // wait result
	                IF "DB_executeQuery".dataReady THEN
	                    "DB_executeQuery".readyForNextQuery := TRUE;

	                    #Dispatcher["updatePartOnMC"] := 0;
	                END_IF;

	            31..35: // prelievo PALLET da macchina -> POS_PLANT=1000
	                // stesso difetto e stessa correzione del 21..25: si esce dal
	                // proprio range prima di mettersi in attesa del ponte.
	                //
	                // IL PALLET E' QUELLO IN MACCHINA, NON QUELLO DELL'ORDINE (18/9).
	                // In automatico si leggeva order.PALLET, che a FINE PRODUZIONE
	                // vale zero: l'ordine e' chiuso o riallineato, e la UPDATE usciva
	                // con WHERE ID=0 senza toccare niente. Il pallet restava a
	                // POS_PLANT=101 (in macchina) mentre era in pinza, e il sistema
	                // non sapeva piu' dov'era. Visto in campo smontando il pallet 9 a
	                // produzione conclusa.
	                // Il registro DB_MC1.pallet dice cosa c'era fisicamente dentro, ed
	                // e' l'unica fonte valida qui: e' lo stesso registro che il 60
	                // azzera subito dopo, proprio perche' il pallet e' uscito.
	                IF "SqlCommands".sqlCommands[0] = '' THEN
	                    IF NOT #RemoteMode THEN
	                        #pieceReq := #PalletRequested;
	                    ELSIF #MCRequested = 2 THEN
	                        #pieceReq := "DB_MC2".pallet;
	                    ELSE
	                        #pieceReq := "DB_MC1".pallet;
	                    END_IF;
	                    #queryTemp := CONCAT(IN1 := 'UPDATE POSITION SET STATUS=',
	                                         IN2 := "INT_TO_STRING_WITHOUT_SIGN"(#Dispatcher["updatePartOnMC"] - 30),
	                                         IN3 := ' WHERE PARENT like $'MC_',
	                                         IN4 := "INT_TO_STRING_WITHOUT_SIGN"(#MCRequested),
	                                         IN5 := '%$' AND PARENT NOT LIKE $'%pallet%$'; UPDATE Pallet SET POS_PLANT=1000 WHERE ID=',
	                                         IN6 := "INT_TO_STRING_WITHOUT_SIGN"(#pieceReq));
	                    #queryStartExecution := TRUE;
	                    #Dispatcher["updatePartOnMC"] := 36;
	                END_IF;

	            36:  // attesa presa in carico della query pallet (stato fuori dai range)
	                IF NOT "DB_executeQuery".readyForNextQuery THEN
	                    #Dispatcher["updatePartOnMC"] := 30;
	                END_IF;
	        END_CASE;
	    END_REGION

	    REGION updatePartOnTray
	        //Activated with dispatcher=10+statusPart (RAW,FINISHED)
	        CASE #Dispatcher["updatePartOnTray"] OF
	            0:  // nothing to do
	                ;

	            12: // Update DB with EMPTY part
	                // MC1 E' IL DEFAULT (18/9): vedi la nota estesa al 15. La forma
	                // "IF MCRequested = 1 THEN MC1 ELSE MC2" prende DB_MC2.order.ID —
	                // sempre zero in questa cella — ogni volta che MCRequested non e'
	                // esattamente 1, e il 95 substate 0 di FB204 lo azzera prima di
	                // lanciare il deposito. Qui #temp non finisce in nessuna query,
	                // quindi non fa danni: si allinea per non lasciare tre forme
	                // diverse nello stesso blocco.
	                IF #MCRequested = 2 THEN
	                    #temp := DINT_TO_INT("DB_MC2".order.ID);
	                ELSE
	                    #temp := DINT_TO_INT("DB_MC1".order.ID);
	                END_IF;

	                IF "SqlCommands".sqlCommands[0] = '' THEN
	                    // UGUAGLIANZA, NON LIKE (16/9): 'TRAY_1%' prendeva anche TRAY_10,
	                    // TRAY_11 e TRAY_12 -> quattro cassetti aggiornati insieme. Con i
	                    // cassetti 1-9 il difetto era invisibile; con l'1 in gioco insieme
	                    // ai due cifre ha riscritto TRAY_1 e TRAY_12 in parallelo.
	                    IF NOT #RemoteMode AND #PartSubPos > 0 THEN   // HMI: posizione esatta, nessun ordine
	                        #queryTemp := CONCAT(IN1 := 'UPDATE [POSITION] SET STATUS=2 WHERE PARENT=$'TRAY_',
	                                             IN2 := "INT_TO_STRING_WITHOUT_SIGN"(#Tray_ID),
	                                             IN3 := '$' AND SUB_POS=',
	                                             IN4 := "INT_TO_STRING_WITHOUT_SIGN"(#PartSubPos));
	                        #queryStartExecution := TRUE;

	                        #Dispatcher["updatePartOnTray"] := 20;
	                    ELSE
	                        // AUTOMATICO: svuota la tasca da cui il robot ha appena prelevato
	                        // (SUB_POS congelato), non la prima con un grezzo.
	                        #queryTemp := CONCAT(IN1 := 'UPDATE [POSITION] SET STATUS=2 WHERE PARENT=$'TRAY_',
	                                             IN2 := "INT_TO_STRING_WITHOUT_SIGN"(#Tray_ID),
	                                             IN3 := '$' AND SUB_POS=',
	                                             IN4 := "INT_TO_STRING_WITHOUT_SIGN"(#PartSubPos));
	                        #queryStartExecution := TRUE;

	                        #Dispatcher["updatePartOnTray"] := 20;
	                    END_IF;
	                END_IF;

	            15: // Update DB with FINISHED part
	                // MC1 E' IL DEFAULT (18/9). La forma "IF MCRequested = 1 THEN MC1
	                // ELSE MC2" leggeva DB_MC2.order.ID — che in questa cella vale
	                // SEMPRE zero — ogni volta che MCRequested non era esattamente 1.
	                // E il 95 substate 0 di FB204 lo AZZERA prima di lanciare il
	                // deposito del finito:
	                //     "DB_Robot".MissionCode := "MISSION_UnloadPartFromRobot";
	                //     "DB_Robot".MCRequested := 0;
	                // Quindi #temp usciva a zero proprio sul percorso del ciclo a
	                // missione 16, e con lui sia Order_ID sulla tasca sia il
	                // congelamento di OrderIdMC.
	                // Visto in campo sul 1102: pezzi alternati, uno con Order_ID
	                // corretto (deposito dal 52/58, dove MCRequested resta a 1) e uno
	                // con zero (deposito dal 95 substate 0).
	                IF #MCRequested = 2 THEN
	                    #temp := DINT_TO_INT("DB_MC2".order.ID);
	                ELSE
	                    #temp := DINT_TO_INT("DB_MC1".order.ID);
	                END_IF;

	                IF "SqlCommands".sqlCommands[0] = '' THEN
	                    IF NOT #RemoteMode AND #PartSubPos > 0 THEN   // HMI: posizione esatta; il pezzo torna com'era (RAW)
	                        #queryTemp := CONCAT(IN1 := 'UPDATE [POSITION] SET STATUS=4 WHERE PARENT=$'TRAY_',
	                                             IN2 := "INT_TO_STRING_WITHOUT_SIGN"(#Tray_ID),
	                                             IN3 := '$' AND SUB_POS=',
	                                             IN4 := "INT_TO_STRING_WITHOUT_SIGN"(#PartSubPos));
	                        #queryStartExecution := TRUE;

	                        #Dispatcher["updatePartOnTray"] := 20;
	                    ELSE
	                        // AUTOMATICO: marca finita la tasca del grezzo entrato in macchina
	                        // (PartSubPosMC), non quella del grezzo prelevato per il ciclo dopo.
	                        //
	                        // ORDER_ID SCRITTO QUI (18/9): fino a oggi lo scriveva SOLO il
	                        // comando 39 dal pannello, alla dichiarazione manuale della
	                        // tasca. Il ciclo automatico cambiava STATUS e lasciava
	                        // Order_ID com'era — zero se nessuno aveva dichiarato, oppure
	                        // dell'ordine PRECEDENTE se la tasca veniva riusata.
	                        // PRODUCTED della vista WORKORDERS conta le tasche a 5
	                        // raggruppate per Order_ID, quindi contava i pezzi dichiarati
	                        // a mano, non quelli prodotti.
	                        //
	                        // SI USA L'ORDINE CONGELATO (OrderIdMC), non quello attivo:
	                        // il pezzo appartiene all'ordine che lo ha LAVORATO, che col
	                        // ciclo a missione 16 puo' non essere piu' quello corrente
	                        // quando il finito torna nel cassetto.
	                        // Ripiego su #temp quando OrderIdMC e' zero: capita al primo
	                        // giro dopo un reinit o un reset, e li' l'ordine corrente e'
	                        // l'unica ipotesi sensata — meglio di perdere il pezzo con
	                        // Order_ID=0, che nessun conteggio vedrebbe.
	                        IF #OrderIdMC > 0 THEN
	                            #declMap := #OrderIdMC;
	                        ELSE
	                            #declMap := #temp;
	                        END_IF;
	                        #queryTemp := CONCAT(IN1 := 'UPDATE [POSITION] SET STATUS=5, Order_ID=',
	                                             IN2 := "INT_TO_STRING_WITHOUT_SIGN"(#declMap),
	                                             IN3 := ' WHERE PARENT=$'TRAY_',
	                                             IN4 := "INT_TO_STRING_WITHOUT_SIGN"(#TrayIdMC),
	                                             IN5 := '$' AND SUB_POS=',
	                                             IN6 := "INT_TO_STRING_WITHOUT_SIGN"(#PartSubPosMC));

	                        // ULTIMO USO di PartSubPosMC, TrayIdMC e OrderIdMC per questo
	                        // pezzo: da qui in poi descrivono il grezzo appena entrato.
	                        // Il congelamento va fatto QUI perche' la missione 16 non
	                        // passa da Part_Robot_to_MC (dove avviene l'altro).
	                        #PartSubPosMC := #PartSubPos;
	                        #TrayIdMC := #Tray_ID;

	                        // L'ORDINE SI CONGELA SOLO SE E' VALIDO: uno zero non
	                        // descrive niente e cancellerebbe il valore buono del giro
	                        // precedente. Cintura in piu' oltre al default MC1 qui sopra.
	                        IF #temp > 0 THEN
	                            #OrderIdMC := #temp;
	                        END_IF;

	                        #queryStartExecution := TRUE;

	                        #Dispatcher["updatePartOnTray"] := 20;
	                    END_IF;
	                END_IF;

	            17: // Update DB with ABORTED part
	                // MC1 E' IL DEFAULT (18/9): vedi la nota al 15.
	                // NB: questo ramo e' CODICE MORTO — updatePartOnTray viene lanciato
	                // solo con 12 (10+EMPTY) e 15 (10+FINISHED), nessuno scrive mai 17.
	                // Resta per quando servira' tracciare gli scarti, ma oggi non gira.
	                IF #MCRequested = 2 THEN
	                    #temp := DINT_TO_INT("DB_MC2".order.ID);
	                ELSE
	                    #temp := DINT_TO_INT("DB_MC1".order.ID);
	                END_IF;

	                IF "SqlCommands".sqlCommands[0] = '' THEN
	                    #queryTemp := CONCAT(IN1 := 'UPDATE [POSITION] SET STATUS=7 WHERE PARENT=$'TRAY_',
	                                         IN2 := "INT_TO_STRING_WITHOUT_SIGN"(#Tray_ID),
	                                         IN3 := '$' AND id in (select top 1 id from position where parent=$'TRAY_',
	                                         IN4 := "INT_TO_STRING_WITHOUT_SIGN"(#Tray_ID),
	                                         IN5 := '$' AND Status=2 ',     //first empty position
	                                         IN6 := 'AND Order_ID=',
	                                         IN7 := "INT_TO_STRING_WITHOUT_SIGN"(#temp),
	                                         IN8 := ')');
	                    #queryStartExecution := TRUE;

	                    #Dispatcher["updatePartOnTray"] := 20;
	                END_IF;

	            20:  // execute query
	                IF NOT "DB_executeQuery".readyForNextQuery THEN
	                    #Dispatcher["updatePartOnTray"] := 30;
	                END_IF;
	            30:  // wait result
	                IF "DB_executeQuery".dataReady THEN
	                    "DB_executeQuery".readyForNextQuery := TRUE;

	                    #Dispatcher["updatePartOnTray"] := 0;
	                END_IF;
	        END_CASE;
	    END_REGION

	    REGION Reset or log mission
	        CASE #Dispatcher["Reset_or_log_MissionData"] OF
	            0: //nothing to do
	                ;
	            10: //reset mission data ***START HERE***
	                "DB_RobotMission"."Command" := 0;
	                "DB_RobotMission"."X_Pick-Place" := 0;
	                "DB_RobotMission"."Y_Pick-Place" := 0;
	                "DB_RobotMission"."Z_Pick-Place" := 0;
	                "DB_RobotMission"."XRot_Pick-Place" := 0;
	                "DB_RobotMission"."YRot_Pick-Place" := 0;
	                "DB_RobotMission"."ZRot_Pick-Place" := 0;
	                "DB_RobotMission"."Gripper_code" := 0;
	                "DB_RobotMission"."Gripper1_XDim" := 0;
	                "DB_RobotMission"."Gripper1_YDim" := 0;
	                "DB_RobotMission"."Gripper1_ZDim" := 0;
	                "DB_RobotMission"."Gripper1_XRotDim" := 0;
	                "DB_RobotMission"."Gripper1_YRotDim" := 0;
	                "DB_RobotMission"."Gripper1_ZRotDim" := 0;
	                "DB_RobotMission".Gripper1_Valve := 0;
	                "DB_RobotMission"."Gripper2_XDim" := 0;
	                "DB_RobotMission"."Gripper2_YDim" := 0;
	                "DB_RobotMission"."Gripper2_ZDim" := 0;
	                "DB_RobotMission"."Gripper2_XRotDim" := 0;
	                "DB_RobotMission"."Gripper2_YRotDim" := 0;
	                "DB_RobotMission"."Gripper2_ZRotDim" := 0;
	                "DB_RobotMission".Gripper2_Valve := 0;
	                "DB_RobotMission"."X_approach" := 0;
	                "DB_RobotMission"."Y_approach" := 0;
	                "DB_RobotMission"."Z_approach" := 0;
	                "DB_RobotMission"."XRot_approach" := 0;
	                "DB_RobotMission"."YRot_approach" := 0;
	                "DB_RobotMission"."ZRot_approach" := 0;
	                "DB_RobotMission"."ApproachType" := 0;
	                "DB_RobotMission"."Unit_code" := 0;
	                "DB_RobotMission"."Object_Type" := 0;
	                "DB_RobotMission"."Gripper_Side" := 0;

	                #Dispatcher["Reset_or_log_MissionData"] := 0;

	            100://save data mission on log DB
	                //prepare mission data ***START HERE***
	                IF "SqlCommands".sqlCommands[0] = '' THEN
	                    IF "DB_RobotMission"."XRot_Pick-Place" = "CMD_RobotChangeDataForGripper" THEN
	                        #queryTemp := CONCAT(IN1 := 'INSERT INTO LOG ([DATA], DESCR, UNIT_A, UNIT_B) VALUES(getDate()',
	                                             IN2 := '$'Robot_MISSION$',',
	                                             IN3 := '$'',
	                                             IN4 := "INT_TO_STRING_WITHOUT_SIGN"(IN := "DB_RobotMission".Command),
	                                             IN5 := '$',',
	                                             IN6 := '$'',
	                                             IN7 := "INT_TO_STRING_WITHOUT_SIGN"(DINT_TO_INT("DB_RobotMission".Gripper1_XDim)),
	                                             IN8 := ', ',
	                                             IN9 := "INT_TO_STRING_WITHOUT_SIGN"(DINT_TO_INT("DB_RobotMission".Gripper1_YDim)),
	                                             IN10 := ', ',
	                                             IN11 := "INT_TO_STRING_WITHOUT_SIGN"(DINT_TO_INT("DB_RobotMission".Gripper1_ZDim)),
	                                             IN12 := ', ',
	                                             IN13 := "INT_TO_STRING_WITHOUT_SIGN"(DINT_TO_INT("DB_RobotMission".Gripper1_XRotDim)),
	                                             IN14 := ', ',
	                                             IN15 := "INT_TO_STRING_WITHOUT_SIGN"(DINT_TO_INT("DB_RobotMission".Gripper1_YRotDim)),
	                                             IN16 := ', ',
	                                             IN17 := "INT_TO_STRING_WITHOUT_SIGN"(DINT_TO_INT("DB_RobotMission".Gripper1_ZRotDim)),
	                                             IN18 := ', ',
	                                             IN19 := "INT_TO_STRING_WITHOUT_SIGN"(DINT_TO_INT("DB_RobotMission".Gripper2_XDim)),
	                                             IN20 := ', ',
	                                             IN21 := "INT_TO_STRING_WITHOUT_SIGN"(DINT_TO_INT("DB_RobotMission".Gripper2_YDim)),
	                                             IN22 := ', ',
	                                             IN23 := "INT_TO_STRING_WITHOUT_SIGN"(DINT_TO_INT("DB_RobotMission".Gripper2_ZDim)),
	                                             IN24 := ', ',
	                                             IN25 := "INT_TO_STRING_WITHOUT_SIGN"(DINT_TO_INT("DB_RobotMission".Gripper2_XRotDim)),
	                                             IN26 := ', ',
	                                             IN27 := "INT_TO_STRING_WITHOUT_SIGN"(DINT_TO_INT("DB_RobotMission".Gripper2_YRotDim)),
	                                             IN28 := ', ',
	                                             IN29 := "INT_TO_STRING_WITHOUT_SIGN"(DINT_TO_INT("DB_RobotMission".Gripper2_ZRotDim)),
	                                             IN30 := '$'');
	                    ELSE
	                        #queryTemp := CONCAT(IN1 := 'INSERT INTO LOG ([DATA], DESCR, UNIT_A, UNIT_B) VALUES(getDate()',
	                                             IN2 := '$'Robot_MISSION$',',
	                                             IN3 := '$'',
	                                             IN4 := "INT_TO_STRING_WITHOUT_SIGN"(IN := "DB_RobotMission".Command),
	                                             IN5 := '$',',
	                                             IN6 := '$'',
	                                             IN7 := "INT_TO_STRING_WITHOUT_SIGN"(DINT_TO_INT("DB_RobotMission"."X_Pick-Place")),
	                                             IN8 := ', ',
	                                             IN9 := "INT_TO_STRING_WITHOUT_SIGN"(DINT_TO_INT("DB_RobotMission"."Y_Pick-Place")),
	                                             IN10 := ', ',
	                                             IN11 := "INT_TO_STRING_WITHOUT_SIGN"(DINT_TO_INT("DB_RobotMission"."Z_Pick-Place")),
	                                             IN12 := ', ',
	                                             IN13 := "INT_TO_STRING_WITHOUT_SIGN"(DINT_TO_INT("DB_RobotMission"."XRot_Pick-Place")),
	                                             IN14 := ', ',
	                                             IN15 := "INT_TO_STRING_WITHOUT_SIGN"(DINT_TO_INT("DB_RobotMission"."YRot_Pick-Place")),
	                                             IN16 := ', ',
	                                             IN17 := "INT_TO_STRING_WITHOUT_SIGN"(DINT_TO_INT("DB_RobotMission"."ZRot_Pick-Place")),
	                                             IN18 := ', ',
	                                             IN19 := "INT_TO_STRING_WITHOUT_SIGN"(DINT_TO_INT("DB_RobotMission".ApproachType)),
	                                             IN20 := ', ',
	                                             IN21 := "INT_TO_STRING_WITHOUT_SIGN"(DINT_TO_INT("DB_RobotMission".Unit_code)),
	                                             IN22 := ', ',
	                                             IN23 := "INT_TO_STRING_WITHOUT_SIGN"(DINT_TO_INT("DB_RobotMission".X_approach)),
	                                             IN24 := ', ',
	                                             IN25 := "INT_TO_STRING_WITHOUT_SIGN"(DINT_TO_INT("DB_RobotMission".Y_approach)),
	                                             IN26 := ', ',
	                                             IN27 := "INT_TO_STRING_WITHOUT_SIGN"(DINT_TO_INT("DB_RobotMission".Z_approach)),
	                                             IN28 := ', ',
	                                             IN29 := "INT_TO_STRING_WITHOUT_SIGN"(DINT_TO_INT("DB_RobotMission".Object_Type)),
	                                             IN30 := ', ');

	                        #queryTemp := CONCAT(IN1 := #queryTemp,
	                                             IN2 := "INT_TO_STRING_WITHOUT_SIGN"(DINT_TO_INT("DB_RobotMission".Gripper_Side)),
	                                             IN3 := ', ',
	                                             IN4 := "INT_TO_STRING_WITHOUT_SIGN"(DINT_TO_INT("DB_RobotMission".Object_Type)),
	                                             IN5 := '$'');
	                    END_IF;
	                    #queryStartExecution := TRUE;

	                    #Dispatcher["Reset_or_log_MissionData"] := 115;
	                END_IF;
	            115:  //execute query
	                IF NOT "DB_executeQuery".dataReady THEN
	                    #Dispatcher["Reset_or_log_MissionData"] := 120;
	                END_IF;

	            120: //wait anwser
	                IF "DB_executeQuery".dataReady THEN //AND NOT "DB_executeQuery".dataError
	                    #Dispatcher["Reset_or_log_MissionData"] := 0;
	                    (*ELSIF "DB_executeQuery".dataError THEN
	                        //Error
	                        #Error := 999;
	                        #Dispatcher["Reset_or_log_MissionData"] := 99;
	                        *)
	                END_IF;

	        END_CASE;
	    END_REGION

	    REGION Declare_Position
	        CASE #Dispatcher["_Declare_Position"] OF
	            0:  // nothing to do
	                ;
	            10: // UPDATE della singola tasca del cassetto estratto.
	                // Order_ID all'ordine attivo per lo stato 4 (grezzo): senza, la
	                // tasca non verrebbe mai vista dalle query del ciclo automatico.
	                // UGUAGLIANZA, NON LIKE (16/9): con il LIKE il cassetto 1 avrebbe
	                // aggiornato anche 10, 11 e 12.
	                IF "SqlCommands".sqlCommands[0] = '' THEN
	                    #queryTemp := CONCAT(IN1 := 'UPDATE [POSITION] SET STATUS=',
	                                         IN2 := "INT_TO_STRING_WITHOUT_SIGN"(#declStato),
	                                         IN3 := ', Order_ID=',
	                                         IN4 := "INT_TO_STRING_WITHOUT_SIGN"(DINT_TO_INT("DB_MC1".order.ID)),
	                                         IN5 := ' WHERE PARENT=$'TRAY_',
	                                         IN6 := "INT_TO_STRING_WITHOUT_SIGN"("DB_BOX_1".ExtractedTray),
	                                         IN7 := '$' AND SUB_POS=',
	                                         IN8 := "INT_TO_STRING_WITHOUT_SIGN"(#declSubPos));
	                    #queryStartExecution := TRUE;
	                    #Dispatcher["_Declare_Position"] := 20;
	                END_IF;

	            15: // TIPO PEZZO dell'intero cassetto estratto (comando 44).
	                // Un cassetto contiene un solo tipo, quindi si dichiara in blocco:
	                // dichiararlo tasca per tasca sarebbe dodici click e l'operatore
	                // smetterebbe di farlo. Part_Type e' il campo che decide cosa il
	                // robot va a prendere (16/9), quindi vale per tutte le tasche.
	                IF "SqlCommands".sqlCommands[0] = '' THEN
	                    #queryTemp := CONCAT(IN1 := 'UPDATE [POSITION] SET Part_Type=',
	                                         IN2 := "INT_TO_STRING_WITHOUT_SIGN"(#declTipo),
	                                         IN3 := ' WHERE PARENT=$'TRAY_',
	                                         IN4 := "INT_TO_STRING_WITHOUT_SIGN"("DB_BOX_1".ExtractedTray),
	                                         IN5 := '$'');
	                    #queryStartExecution := TRUE;
	                    #Dispatcher["_Declare_Position"] := 20;
	                END_IF;

	            20:  // presa in carico VERIFICATA: SqlData e il ponte sono condivisi,
	                // non basta che il ponte sia occupato — deve esserci LA NOSTRA
	                // query, altrimenti il 30 chiude sulla risposta di un altro
	                // richiedente e l'UPDATE della tasca non e' mai partito.
	                IF NOT "DB_executeQuery".readyForNextQuery
	                    AND "SqlCommands".sqlCommands[0] = #queryTemp THEN
	                    #Dispatcher["_Declare_Position"] := 30;
	                END_IF;

	            30:  // wait result
	                IF "DB_executeQuery".dataReady THEN
	                    "DB_executeQuery".readyForNextQuery := TRUE;
	                    IF #declTipo > 0 THEN
	                        "FC_MQTT"(insert := true,
	                                  send := false,
	                                  topic := 'FROM_PLANT/DECLARE/TRAYTYPE',
	                                  payload := STRING_TO_WSTRING(CONCAT(IN1 := "INT_TO_STRING_WITHOUT_SIGN"("DB_BOX_1".ExtractedTray),
	                                                                                                   IN2 := ';',
	                                                                                                   IN3 := "INT_TO_STRING_WITHOUT_SIGN"(#declTipo))));
	                        #declTipo := 0;
	                    ELSE
	                        "FC_MQTT"(insert := true,
	                                  send := false,
	                                  topic := 'FROM_PLANT/DECLARE/TRAY',
	                                  payload := STRING_TO_WSTRING(CONCAT(IN1 := "INT_TO_STRING_WITHOUT_SIGN"("DB_BOX_1".ExtractedTray),
	                                                                                                   IN2 := ';',
	                                                                                                   IN3 := "INT_TO_STRING_WITHOUT_SIGN"(#declSubPos),
	                                                                                                   IN4 := ';',
	                                                                                                   IN5 := "INT_TO_STRING_WITHOUT_SIGN"(#declStato))));
	                    END_IF;
	                    #Dispatcher["_Declare_Position"] := 0;
	                ELSIF "DB_executeQuery".dataError THEN
	                    #Error := 20007;
	                    #declTipo := 0;
	                    "DB_executeQuery".readyForNextQuery := TRUE;
	                    #Dispatcher["_Declare_Position"] := 0;
	                END_IF;
	        END_CASE;
	    END_REGION

	END_REGION

	REGION Declare_State
	    CASE #Dispatcher["_Declare_State"] OF
	        0: //nothing to do
	            ;
	        10: // tabula rasa (indice 31 escluso dal reset per costruzione)
	            #RESET_ALL_DISPATCH := TRUE;
	            #Dispatcher["_Declare_State"] := 15;
	        15: // validazione presenza pinza vs sensore
	            IF (#declGripper > 0) XOR "Gripper_mounted" THEN
	                #Error := 945;   // dichiarazione incoerente col sensore pinza
	                #Dispatcher["_Declare_State"] := 945;
	            ELSIF #declCont1 = 3 AND #declCont2 = 3 THEN
	                #Error := 944;   // pallet dichiarato su entrambi i lati: impossibile
	                #Dispatcher["_Declare_State"] := 944;
	            ELSIF #declGripper = 0 THEN
	                // flangia nuda dichiarata e confermata: azzera e chiudi
	                #Gripper_ID[1] := 0;
	                #Gripper_ID[2] := 0;
	                #GripperOccuped[1] := FALSE;
	                #GripperOccuped[2] := FALSE;
	                #Dispatcher["updateGripperOnRobot"] := 10;
	                #Dispatcher["_Declare_State"] := 70;
	            ELSE
	                #Dispatcher["_Declare_State"] := 20;
	            END_IF;
	        20: // query lato 2 (gemella sullo stesso SUB_POS; include se stessa per garantire >=1 riga)
	            // Serve QUI solo per VALIDARE declCont2: la scrittura dei registri la
	            // fa la catena unica al 40.
	            IF "SqlCommands".sqlCommands[0] = '' THEN
	                #queryTemp := CONCAT(IN1 := 'select ID from GRIPPER where ID=',
	                                     IN2 := "INT_TO_STRING_WITHOUT_SIGN"(#declGripper),
	                                     IN3 := ' or (SUB_POS>0 and SUB_POS in (select SUB_POS from GRIPPER where ID=',
	                                     IN4 := "INT_TO_STRING_WITHOUT_SIGN"(#declGripper),
	                                     IN5 := '))');
	                #queryStartExecution := TRUE;
	                #Dispatcher["_Declare_State"] := 25;
	            END_IF;
	        25: // presa in carico query (pattern FB204: conferma che in [0] c'e' LA NOSTRA query)
	            IF NOT "DB_executeQuery".readyForNextQuery
	                AND "SqlCommands".sqlCommands[0] = #queryTemp THEN
	                #Dispatcher["_Declare_State"] := 30;
	            END_IF;
	        30: // validazione: il lato 2 dichiarato esiste davvero?
	            IF "DB_executeQuery".dataReady AND "DB_executeQuery".noData THEN
	                // pinza dichiarata inesistente a DB: con FB6 corretto "zero righe"
	                // non e' piu' dataError, va intercettato qui.
	                "DB_executeQuery".readyForNextQuery := TRUE;
	                #Error := 946;   // errore DB in dichiarazione
	                #Dispatcher["_Declare_State"] := 946;
	            ELSIF "DB_executeQuery".dataReady AND NOT "DB_executeQuery".dataError THEN
	                IF "SqlData".data.rowCount <= 1 AND #declCont2 > 0 THEN
	                    "DB_executeQuery".readyForNextQuery := TRUE;
	                    #Error := 944;   // contenuto dichiarato su lato inesistente
	                    #Dispatcher["_Declare_State"] := 944;
	                ELSE
	                    "DB_executeQuery".readyForNextQuery := TRUE;
	                    #queryTemp := '';
	                    #queryStartExecution := FALSE;
	                    #GripperOccuped[1] := #declCont1 > 0;
	                    #GripperOccuped[2] := #declCont2 > 0;
	                    #Dispatcher["_Declare_State"] := 40;
	                END_IF;
	            ELSIF "DB_executeQuery".dataError THEN
	                "DB_executeQuery".readyForNextQuery := TRUE;
	                #Error := 946;   // errore DB in dichiarazione
	                #Dispatcher["_Declare_State"] := 946;
	            END_IF;
	        40: // registri + database alla catena unica (17/9)
	            #GripperRequested := #declGripper;
	            #Dispatcher["_Set_Gripper_OnBoard"] := 10;
	            #Dispatcher["_Declare_State"] := 45;
	        45:
	            IF #Dispatcher["_Set_Gripper_OnBoard"] = 0 THEN
	                #Dispatcher["get_TCP_Data"] := 10;
	                #Dispatcher["_Declare_State"] := 50;
	            END_IF;
	        50: // TCP aggiornato al robot
	            IF #Dispatcher["get_TCP_Data"] = 0 THEN
	                #Dispatcher["_Declare_State"] := 55;
	            END_IF;
	        55: // stato lato 1
	            CASE #declCont1 OF
	                1:
	                    #declMap := DINT_TO_INT("RAW");
	                2:
	                    #declMap := DINT_TO_INT("FINISHED");
	                3:
	                    // PALLET: RAW come il resto del sistema (18/9). LOADED=1 non e'
	                    // interrogato da nessuna vista ne' da nessun filtro del ciclo,
	                    // che cercano tutti STATUS=4: un pallet dichiarato LOADED era
	                    // invisibile. Il 50 di Pallet_TRAY_to_Robot lo scrive RAW da
	                    // sempre — "il pallet lo considero grezzo cosi' va in macchina".
	                    #declMap := DINT_TO_INT("RAW");
	                ELSE
	                    #declMap := DINT_TO_INT("EMPTY");
	            END_CASE;
	            "DB_RobotMission".Gripper_Side := 1;
	            #Dispatcher["updatePartOnRobot"] := 10 + #declMap;
	            #Dispatcher["_Declare_State"] := 60;
	        60:
	            IF #Dispatcher["updatePartOnRobot"] = 0 THEN
	                IF #Gripper_ID[2] > 0 THEN
	                    CASE #declCont2 OF
	                        1:
	                            #declMap := DINT_TO_INT("RAW");
	                        2:
	                            #declMap := DINT_TO_INT("FINISHED");
	                        3:
	                            // pallet: RAW, vedi nota al 55
	                            #declMap := DINT_TO_INT("RAW");
	                        ELSE
	                            #declMap := DINT_TO_INT("EMPTY");
	                    END_CASE;
	                    #Dispatcher["updatePartOnRobot"] := 20 + #declMap;
	                    #Dispatcher["_Declare_State"] := 65;
	                ELSE
	                    #Dispatcher["_Declare_State"] := 68;
	                END_IF;
	            END_IF;
	        65:
	            IF #Dispatcher["updatePartOnRobot"] = 0 THEN
	                #Dispatcher["_Declare_State"] := 68;
	            END_IF;
	        68: // pallet a bordo -> POS_PLANT=1000
	            IF #declCont1 = 3 OR #declCont2 = 3 THEN
	                IF "SqlCommands".sqlCommands[0] = '' THEN
	                    IF #declCont1 = 3 THEN
	                        #declMap := #declId1;
	                    ELSE
	                        #declMap := #declId2;
	                    END_IF;
	                    #queryTemp := CONCAT(IN1 := 'UPDATE Pallet SET POS_PLANT=1000 WHERE ID=',
	                                         IN2 := "INT_TO_STRING_WITHOUT_SIGN"(#declMap));
	                    #queryStartExecution := TRUE;
	                    #Dispatcher["_Declare_State"] := 69;
	                END_IF;
	            ELSE
	                #Dispatcher["_Declare_State"] := 70;
	            END_IF;
	        69:
	            IF NOT "DB_executeQuery".readyForNextQuery THEN
	                #Dispatcher["_Declare_State"] := 695;
	            END_IF;
	        695:
	            IF "DB_executeQuery".dataReady THEN
	                "DB_executeQuery".readyForNextQuery := TRUE;
	                #Dispatcher["_Declare_State"] := 70;
	            END_IF;
	        70: // chiusura + riepilogo
	            IF #Dispatcher["updateGripperOnRobot"] = 0 THEN
	                "FC_MQTT"(insert := true,
	                          send := false,
	                          topic := 'FROM_PLANT/DECLARE/ROBOT',
	                          payload := STRING_TO_WSTRING(CONCAT(IN1 := "INT_TO_STRING_WITHOUT_SIGN"(#Gripper_ID[1]),
	                                                                                           IN2 := ';',
	                                                                                           IN3 := "INT_TO_STRING_WITHOUT_SIGN"(#declCont1),
	                                                                                           IN4 := ';',
	                                                                                           IN5 := "INT_TO_STRING_WITHOUT_SIGN"(#declCont2))));
	                #MissionCode := 0;
	                #Dispatcher["_Declare_State"] := 0;
	            END_IF;
	        944:
	            ; // contenuto su lato inesistente
	        945:
	            ; // incoerenza sensore pinza
	        946:
	            ; // errore DB
	    END_CASE;
	END_REGION

	REGION execute query
	    // IF "DB_executeQuery".dataReady AND "DB_executeQuery".readyForNextQuery THEN
	    (*
	    "DB_executeQuery"(query := #queryTemp,
	                      params := #paramsTemp,
	                      exec := #queryStartExecution);
	    #queryStartExecution := false;
	    //#queryTemp := '';
	 *)
	 // END_IF;
	END_REGION

	REGION updateHMI
	    //inconsistency datas and sensors
	    IF "DB_RobotMissionStatus".StatusCode = "cmd_waitingNewCmd" AND
	        (
	        (#GripperOccuped[1] XOR "DB_RobotMissionStatus".StatusRegister.Gripper1_occuped) OR
	        (#GripperOccuped[2] XOR "DB_RobotMissionStatus".StatusRegister.Gripper2_occuped)
	        ) THEN
	        IF NOT #checkInconsistenceFailed THEN
	            "FC_MQTT"(insert := true,
	                      send := false,
	                      topic := 'FROM_PLANT/ALARM/ROBOT',
	                      payload := STRING_TO_WSTRING("INT_TO_STRING_WITHOUT_SIGN"(23)));
	            #checkInconsistenceFailed := true;
	        END_IF;
	    ELSE
	        #checkInconsistenceFailed := false;
	    END_IF;

	    //Mission
	    IF (#MissionCode <> #lastMission) THEN
	        "FC_MQTT"(insert := true,
	                  send := false,
	                  topic := 'FROM_PLANT/LOG/MISSION/ROBOT',
	                  payload := STRING_TO_WSTRING("INT_TO_STRING_WITHOUT_SIGN"(#MissionCode)));

	        #lastMission := #MissionCode;

	        //change description of robot mission
	        IF #Dispatcher["_Gripper_TRAY_to_Robot"] > 0 THEN
	            "FC_MQTT"(insert := true,
	                      send := false,
	                      topic := 'FROM_PLANT/DESCR/ROBOT',
	                      payload := STRING_TO_WSTRING('Drop Gripper'));
	        ELSIF #Dispatcher["_Gripper_Robot_to_TRAY"] > 0 THEN
	            "FC_MQTT"(insert := true,
	                      send := false,
	                      topic := 'FROM_PLANT/DESCR/ROBOT',
	                      payload := STRING_TO_WSTRING('Pick Gripper'));
	        ELSIF #Dispatcher["_Pallet_TRAY_to_Robot"] > 0 THEN
	            "FC_MQTT"(insert := true,
	                      send := false,
	                      topic := 'FROM_PLANT/DESCR/ROBOT',
	                      payload := STRING_TO_WSTRING('Pick Pallet'));
	        ELSIF #Dispatcher["_Pallet_Robot_to_TRAY"] > 0 THEN
	            "FC_MQTT"(insert := true,
	                      send := false,
	                      topic := 'FROM_PLANT/DESCR/ROBOT',
	                      payload := STRING_TO_WSTRING('Drop Pallet'));
	        ELSIF #Dispatcher["_Pallet_MC_to_Robot"] > 0 THEN
	            "FC_MQTT"(insert := true,
	                      send := false,
	                      topic := 'FROM_PLANT/DESCR/ROBOT',
	                      payload := STRING_TO_WSTRING('Pick Pallet from MC'));
	        ELSIF #Dispatcher["_Pallet_Robot_to_MC"] > 0 THEN
	            "FC_MQTT"(insert := true,
	                      send := false,
	                      topic := 'FROM_PLANT/DESCR/ROBOT',
	                      payload := STRING_TO_WSTRING('Drop Pallet on MC'));
	        ELSIF #Dispatcher["_Part_TRAY_to_Robot"] > 0 THEN
	            "FC_MQTT"(insert := true,
	                      send := false,
	                      topic := 'FROM_PLANT/DESCR/ROBOT',
	                      payload := STRING_TO_WSTRING('Pick Part'));
	        ELSIF #Dispatcher["_Part_Robot_to_TRAY"] > 0 THEN
	            "FC_MQTT"(insert := true,
	                      send := false,
	                      topic := 'FROM_PLANT/DESCR/ROBOT',
	                      payload := STRING_TO_WSTRING('Drop Part'));
	        ELSIF #Dispatcher["_Part_Robot_to_MC"] > 0 THEN
	            "FC_MQTT"(insert := true,
	                      send := false,
	                      topic := 'FROM_PLANT/DESCR/ROBOT',
	                      payload := STRING_TO_WSTRING('Drop Part on Machine'));
	        ELSIF #Dispatcher["_Part_MC_to_Robot"] > 0 THEN
	            "FC_MQTT"(insert := true,
	                      send := false,
	                      topic := 'FROM_PLANT/DESCR/ROBOT',
	                      payload := STRING_TO_WSTRING('Pick Part from Machine'));
	        ELSIF #Dispatcher["_Declare_Position"] > 0 THEN
	            "FC_MQTT"(insert := true,
	                      send := false,
	                      topic := 'FROM_PLANT/DESCR/ROBOT',
	                      payload := STRING_TO_WSTRING('Declare Tray Position'));
	        ELSIF #Dispatcher["Extract_TRAY"] > 0 OR #Dispatcher["Extract_TRAY_HMI"] > 0 THEN
	            "FC_MQTT"(insert := true,
	                      send := false,
	                      topic := 'FROM_PLANT/DESCR/ROBOT',
	                      payload := STRING_TO_WSTRING('Extract Tray'));
	        ELSIF #Dispatcher["Release_TRAY"] > 0 OR #Dispatcher["Release_TRAY_HMI"] > 0 THEN
	            "FC_MQTT"(insert := true,
	                      send := false,
	                      topic := 'FROM_PLANT/DESCR/ROBOT',
	                      payload := STRING_TO_WSTRING('Release Tray'));
	        ELSIF #MissionCode = "MISSION_SwapGripper" THEN
	            "FC_MQTT"(insert := true,
	                      send := false,
	                      topic := 'FROM_PLANT/DESCR/ROBOT',
	                      payload := STRING_TO_WSTRING('Swap Gripper'));
	        ELSE
	            "FC_MQTT"(insert := true,
	                      send := false,
	                      topic := 'FROM_PLANT/DESCR/ROBOT',
	                      payload := STRING_TO_WSTRING(''));
	        END_IF;

	    END_IF;

